# B&R Automation Studio project DevOpsDemo
Automation Studio 6.7.1.5; technology packages: mappMotion 6.7.2, mappView 6.7.0, OpcUaCs 6.6.1

## Configuration Config1

CPU X20CP0484, AutomationRuntime 6.7.5, Build 11.3.0

CPU X20CP1686X, AutomationRuntime 6.7.6, Build 11.3.0

### Task classes (Cpu.sw)
```
Cyclic#1 (cycle 1000 us, tolerance 0 us):
  Program <- Program.prg
  RevInfo <- RevInfo.RevInfo.prg
```

### Task classes (Cpu.sw)
```
Cyclic#1 (cycle 1000 us, tolerance 0 us):
  Main <- Main.Main.prg
  EM_Conveyo <- EM_Conveyor.EM_Conveyor.prg
  EM_Filler <- EM_Filler.EM_Filler.prg
  EM_Capper <- EM_Capper.EM_Capper.prg
Cyclic#3 (cycle 50000 us, tolerance 50000000 us):
  Update <- Services.Update.prg
  RevInfo <- RevInfo.RevInfo.prg
Binaries: udbdef, FWRules, TCData, sysconf, iomap, ashwd, BRRole, asfw, arconfig, ashwac, UaCsConfig
Libraries: MpBase, UaCore, AsIecCon, ArProject, runtime, FileIO, sys_lib, brsystem, BrdkPackML, PackMLCore, MpAlarmX, astime, McBase, McAxis, MpAxis, McAcpAx, McAcpPar, standard, AsIODiag, MpServer
```

### Hardware
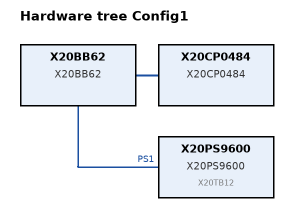
```
X20BB62 : X20BB62 v1.3.0.0
X20CP0484 : X20CP0484 v1.9.0.0  [SL -> X20BB62.SL1]
  Connector IF2:
    ActivateDevice = 1
    Mode = Manual
    InternetAddress = 192.168.2.11
    SubnetMask = 255.255.255.0
    ActivateSnmp = 2
  ConfigurationID = DevOpsDemo_Config1
  UserPartitionSize = 100
  Simulation = 1
  TimerDeviceType = SWIOTIMER
  CyclicTaskClassCount = 3
  Cyclic1Duration = 1000
  Cyclic1Tolerance = 0
  Cyclic2Duration = 5000
  Cyclic2Tolerance = 0
  Cyclic3Duration = 50000
  Cyclic3Tolerance = 50000000
  Cyclic4Duration = 100000
  Cyclic4Tolerance = 100000
  Cyclic5Duration = 200000
  Cyclic5Tolerance = 200000
  Cyclic6Duration = 500000
  Cyclic6Tolerance = 500000
  Cyclic7Duration = 1000000
  Cyclic7Tolerance = 1000000
  Cyclic8Duration = 10000
  Cyclic8Tolerance = 30000000
  FileDevice1
  FileDeviceName1 = USER
  FileDevicePath1 = USER_PATH
  ActivateWebServer = 1
  WebServerProtocol = 1
  ActivateSdm = 1
  Authentication = 0
  ConfigVersion = 0.0.4
X20PS9600 : X20PS9600 v1.6.2.0  [PS -> X20BB62.PS1; SS1 -> X20TB12.SS]
X20TB12 : X20TB12 v1.0.0.0
```

### Config_1.axis - X20CP0484/mappMotion/Config_1.axis
```
Element gAxis_Infeed (Type=axis)
  BaseType = Linear
Element gAxis_Capper (Type=axis)
  BaseType = Rotary
Element gAxis_Outfeed (Type=axis)
  BaseType = Linear
```

### Config.mpbackupcore - X20CP0484/mappServices/Config.mpbackupcore
```
Element gBackupCore (Type=mpbackupcore)
  mapp.Gen:
    Enable = TRUE
    EnableCockpit = FALSE
    Audit = FALSE
    Parent
  Backup:
    AutomaticBackup = Disabled
    AutomaticUpdate = Notify
      DeviceName = UPDATE
      Check = OnEnable
  Alarms = None
```

### Config_1.axis - X20CP1686X/mappMotion/Config_1.axis
```
Element gAxis_Conveyor (Type=axis)
  BaseType = Linear
Element gAxis_Capper (Type=axis)
  MovementLimits:
    Velocity:
      Velocity = 3000
```

## Logical view

Binary libraries used (declarations not repeated): operator, runtime, AsIecCon, MpBase, ArProject, FileIO, sys_lib, brsystem, MpAlarmX, astime, McBase, McAxis, MpAxis, McAcpAx, McAcpPar, standard, AsIODiag, MpServer, AsHttp

### Global.var - Global variables
```iecst
VAR
	gVar : USINT;
END_VAR
```

### Package Logical/Libraries - Global libraries

### Library Logical/Libraries/BrdkPackML (ANSIC, version 3.0.3) - OMAC PackML
Depends on: sys_lib, brsystem

#### BrdkPackML.fun
```iecst
FUNCTION_BLOCK ControlModule (*Control module implementation for OMAC PackML*)
	VAR_INPUT
		Setup : CMSetupType; (*Local setup*) (* *) (*#PAR#;*)
		Interface : CMInterfaceType; (*Publish/Subscribe Interface between Equipment Modules *)
		StateInfo : STRING[255]; (*Status of what the substate is doing or waiting for. Will also be used for logging.*) (* *) (*#CYC#;*)
		State : DINT; (*Control Module state*)
		SubState : DINT := 0; (*The sub state of the module. Can be used for programming the sequence inside a PackML state. Will automatically be reset to 0 by a PackML state change.*) (* *) (*#CYC#;*)
		Continue : BOOL; (*Continue / Acknowledge a state or substate change request when StepMode is enabled*)
	END_VAR
	VAR_OUTPUT
		Info : CMInfoType; (*Additional information about the component*) (* *) (*#CMD#; *)
	END_VAR
	VAR
		Internal : CMInternalType; (*Internal variables*)
	END_VAR
END_FUNCTION_BLOCK

FUNCTION_BLOCK EquipmentModule (*Synchronized PackML state machine handling*) (* $GROUP=mapp Services,$CAT=OMAC PackML,$GROUPICON=Icon_mapp.png,$CATICON=Icon_MpPackML.png *)
	VAR_INPUT
		Setup : EMSetupType; (*Local setup*) (* *) (*#PAR#;*)
		Interface : EMInterfaceType; (*Publish/Subscribe Interface between Equipment Modules *)
		SetModeID : DINT := 1; (*Change the packML mode*)
		StateInfo : STRING[255]; (*Status of what the substate is doing or waiting for. Will also be used for logging.*) (* *) (*#CYC#;*)
		Command : EMCommandType; (*Control commands from ISA-TR88.00.02 commands.*) (* *) (*#CMD#;*)
		SubState : DINT := 0; (*The sub state of the module. Can be used for programming the sequence inside a PackML state. Will automatically be reset to 0 by a PackML state change.*) (* *) (*#CYC#;*)
		Continue : BOOL; (*Continue / Acknowledge a substate change request when StepMode is enabled*)
	END_VAR
	VAR_OUTPUT
		StateCurrent : EMPackMLStateEnum := STATE_UNDEFINED; (*Current state*) (* *) (*#CMD#;*)
		ModeID : EMPackMLModeEnum := MODE_PRODUCTION; (*The current mode*) (* *) (*#CMD#;*)
		Info : EMInfoType; (*Additional information about the component*) (* *) (*#CMD#; *)
	END_VAR
	VAR
		Internal : EMInternalType; (*Internal variables*)
	END_VAR
END_FUNCTION_BLOCK

FUNCTION EMGetModuleAdrByIdx : UDINT (*Returns the address of an Equipment Module on the heap based on the index*)
	VAR_INPUT
		EmIdx : UDINT; (*Index of the Equipment Module*)
	END_VAR
END_FUNCTION

FUNCTION EMGetModuleIdxByName : UDINT (*Returns the index for an Em with the specified name*)
	VAR_INPUT
		EmName : STRING[255]; (*Name of the Equipment Module*)
	END_VAR
END_FUNCTION

FUNCTION EMGetModuleAdrByName : UDINT (*Returns the address of an Equipment Module on the heap based on its name*)
	VAR_INPUT
		EmName : STRING[255]; (*Name of the Equipment Module*)
	END_VAR
END_FUNCTION

FUNCTION EMGetNumberOfModules : UDINT (*Returns the number of Equipment Modules*)
END_FUNCTION

FUNCTION EMGetNumberOfRootModules : UDINT (*Returns the number of root modules. A root module is an Equipment Module with Level 0*)
END_FUNCTION

FUNCTION EMGetWaitingForByIdx : BOOL (*Get WaitingFor from hierarchy index. Returns true on success*)
	VAR_INPUT
		EmIdx : UDINT; (*Index of the root*)
		WaitingFor : EMStatusType; (*EMStatusType*)
	END_VAR
END_FUNCTION

FUNCTION EMGetInterruptedByByIdx : BOOL (*Get InterruptedBy from hierarchy index. Returns true on success*)
	VAR_INPUT
		EmIdx : UDINT; (*Index of the root*)
		InterruptedBy : EMStatusType; (*EMStatusType*)
	END_VAR
END_FUNCTION

FUNCTION EMGetModuleStatus : BOOL (*Get the status from any Equipment Module using the memory address. Returns true on success*)
	VAR_INPUT
		EmAddress : UDINT; (*Address of the Equipment Module*)
		EMStatus : EMStatusType; (*EMStatusType*)
	END_VAR
END_FUNCTION

FUNCTION EMGetModuleStatusByName : BOOL (*Get the status from any Equipment Module using the configured name. Returns true on success*)
	VAR_INPUT
		EmName : STRING[255]; (*Name of the Equipment Module*)
		EMStatus : EMStatusType; (*EMStatusType*)
	END_VAR
END_FUNCTION

FUNCTION EMGetModuleStatusByIdx : BOOL (*Get the status from any Equipment Module using an index. Returns true on success*)
	VAR_INPUT
		EmIdx : UDINT; (*Index of the Equipment Module*)
		EMStatus : EMStatusType; (*EMStatusType*)
	END_VAR
END_FUNCTION

FUNCTION EMGetParentAdr : UDINT (*Returns the address of the parent Equipment Module on the heap*)
	VAR_INPUT
		EmAddress : UDINT; (*Address of the Equipment Module*)
	END_VAR
END_FUNCTION

FUNCTION EMGetChildrenAdrByIdx : UDINT (*Returns the address of a child Equipment Module using an index*)
	VAR_INPUT
		EmAddress : UDINT; (*Address of the Equipment Module*)
		EmIdx : UDINT; (*Index of the child Equipment Module*)
	END_VAR
END_FUNCTION

FUNCTION EMGetSiblingAdrByIdx : UDINT (*Returns the address of a sibling Equipment Module using an index*)
	VAR_INPUT
		EmAddress : UDINT; (*Address of the Equipment Module*)
		EmIdx : UDINT; (*Index of the sibling Equipment Module*)
	END_VAR
END_FUNCTION

FUNCTION EMGetRootAdrByIdx : UDINT (*Returns the address of a root Equipment Module using an index*)
	VAR_INPUT
		EmIdx : UDINT; (*Index of a root Equipment Module*)
	END_VAR
END_FUNCTION

FUNCTION EMGetUserDataAdr : UDINT (*Returns the address of the published userdata from a remote Equipment Module*)
	VAR_INPUT
		EmAddress : UDINT; (*Address of the Equipment Module*)
	END_VAR
END_FUNCTION

FUNCTION EMSetCommand : BOOL (*Send a command to an Equipment Module using its address. Returns true on success*)
	VAR_INPUT
		EmAddress : UDINT; (*Address of the remote Equipment Module to receive the command*)
		EmAddressInterrupter : UDINT; (*Address of the local Equipment Module interrupting the remote Em *)
		Command : EMPackMLCmdEnum; (*Command*)
	END_VAR
END_FUNCTION

FUNCTION EMSetMode : BOOL (*Function changing the mode of an Equipment Module*) (* $GROUP=mapp Services,$CAT=OMAC PackML,$GROUPICON=Icon_mapp.png,$CATICON=Icon_MpPackML.png *)
	VAR_INPUT
		EmAddress : UDINT; (*Address of the target Equipment Module*)
		Mode : DINT; (*Desired mode to change to. The mode must be defined in the mppackmlcore configuration*) (* *) (*#PAR#;*)
	END_VAR
END_FUNCTION

FUNCTION EMSetModeByName : BOOL (*Function changing the mode of an Equipment Module*) (* $GROUP=mapp Services,$CAT=OMAC PackML,$GROUPICON=Icon_mapp.png,$CATICON=Icon_MpPackML.png *)
	VAR_INPUT
		EmName : STRING[255]; (*Name of the target Equipment Module*)
		Mode : DINT; (*Desired mode to change to. *) (* *) (*#PAR#;*)
	END_VAR
END_FUNCTION
```

#### BrdkPackML.typ
```iecst
TYPE
	EMStatusType : 	STRUCT  (*EMStatusType*)
		Name : STRING[255]; (*Em Name*)
		ModeID : UDINT; (*Current Mode*)
		StateCurrent : EMPackMLStateEnum; (*Current State*)
		SubStateCurrent : DINT; (*Current Sub State*)
		StateComplete : BOOL; (*State Complete*)
		StateInfo : STRING[255]; (*Used to describe the action in all states and substates*)
	END_STRUCT;
	EMCommandType : 	STRUCT  (*EMCommandType*)
		Abort : BOOL; (*Go to state Aborting - Can be set in all states except Aborting and Aborted.*)
		Clear : BOOL; (*Go to state Clearing - Can only be set in state Aborted.*)
		Stop : BOOL; (*Go to state Stopping - Can be set in all states except Aborting, Aborted, Clearing, Stopping and Stopped.*)
		Reset : BOOL; (*Go to state Resetting - Can only be set in state Stopped.*)
		Start : BOOL; (*Go to state Starting - Can only be set in state Idle.*)
		Hold : BOOL; (*Go to state Holding. Can only be set in state Execute.*)
		Unhold : BOOL; (*Go to state Unholding. Can only be set in state Held.*)
		Suspend : BOOL; (*Go to state Suspending. Can only be set in state Execute.*)
		Unsuspend : BOOL; (*Go to state Unsuspending. Can only be set in state Suspended.*)
		Complete : BOOL; (*Go to state Completing. Can only be set in state Execute*)
		StateComplete : BOOL; (*Go to next waiting state. Can be set in all acting states and state Execute.*)
	END_STRUCT;
	EMPackMLCmdEnum :
		( (*Command Enum*)
		CMD_UNDEFINED := 0, (*Undefined Command*)
		CMD_RESET := 1, (*PackML Reset Command*)
		CMD_START := 2, (*PackML Start Command*)
		CMD_STOP := 3, (*PackML Stop Command*)
		CMD_HOLD := 4, (*PackML Hold Command*)
		CMD_UNHOLD := 5, (*PackML Unhold Command*)
		CMD_SUSPEND := 6, (*PackML Suspend Command*)
		CMD_UNSUSPEND := 7, (*PackML Unsuspend Command*)
		CMD_ABORT := 8, (*PackML Abort Command*)
		CMD_CLEAR := 9, (*PackML Clear Command*)
		CMD_COMPLETE := 10, (*PackML Complete Command*)
		CMD_SC := 11 (*PackML State Complete Command*)
		);
	EMPackMLModeEnum :
		( (*Mode Enum*)
		MODE_UNDEFINED := 0, (*PackML Undefined mode*)
		MODE_PRODUCTION := 1, (*PackML Production mode*)
		MODE_MAINTENANCE := 2, (*PackML Maintenance mode*)
		MODE_MANUAL := 3, (*PackML Manual mode*)
		MODE_CLEAN := 16, (*PackML Cleaning mode*)
		MODE_JOG := 17, (*PackML Jogging mode*)
		MODE_CIP := 18, (*PackML CIP mode*)
		MODE_CALIBRATION := 19 (*PackML Calibration mode*)
		);
	EMPackMLStateEnum :
		( (*State Enum*)
		STATE_UNDEFINED := 0, (*The system is inactive, no state active*)
		STATE_CLEARING := 1, (*PackML CLEARING state*)
		STATE_STOPPED := 2, (*PackML STOPPED state*)
		STATE_STARTING := 3, (*PackML STARTING state*)
		STATE_IDLE := 4, (*PackML IDLE state*)
		STATE_SUSPENDED := 5, (*PackML SUSPENDED state*)
		STATE_EXECUTE := 6, (*PackML EXECUTE state*)
		STATE_STOPPING := 7, (*PackML STOPPING state*)
		STATE_ABORTING := 8, (*PackML ABORTING state*)
		STATE_ABORTED := 9, (*PackML ABORTED state*)
		STATE_HOLDING := 10, (*PackML HOLDING state*)
		STATE_HELD := 11, (*PackML HELD state*)
		STATE_UNHOLDING := 12, (*PackML UNHOLDING state*)
		STATE_SUSPENDING := 13, (*PackML SUSPENDING state*)
		STATE_UNSUSPENDING := 14, (*PackML UNSUSPENDING state*)
		STATE_RESETTING := 15, (*PackML RESETTING state*)
		STATE_COMPLETING := 16, (*PackML COMPLETING state*)
		STATE_COMPLETED := 17, (*PackML COMPLETED state*)
		STATE_DEACTIVATING := 30, (*Deactivating state. Not a standard PackML state*)
		STATE_DEACTIVATED := 31, (*Deactivated state. Not a standard PackML state*)
		STATE_ACTIVATING := 32 (*Activating state. Not a standard PackML state*)
		);
	EMActivationConditionEnum :
		( (*Activation Enum*)
		ACTIVATE_AUTOMATIC := 0, (*Activate Em automatically when executed*)
		ACTIVATE_BY_PARENT := 1, (*Activate Em if parent is activated*)
		ACTIVATE_BY_PV := 2 (*Activate Em based on PV value*)
		);
	EMSetupType : 	STRUCT  (*EMSetupType*)
		ParentName : STRING[255]; (*Name of the parent. Leave empty is Em is parent at level 0*)
		Name : STRING[255]; (*Name of the Em. If left empty during first execution, the task name is used as Em name*)
		NameIndex : USINT := EM_MAX_NAME_INDEX; (*Index of the Em if having multiple Em's in an array*)
		Activate : BOOL := FALSE; (*PV for ActivationCondition ACTIVATE_BY_PV*)
		ActivationCondition : EMActivationConditionEnum := ACTIVATE_AUTOMATIC; (*Condition for activating the Em*)
		EnableWaitingFor : BOOL := TRUE; (*Enable the WaitingFor log*)
		EnableInterruptedBy : BOOL := TRUE; (*Enable the InterruptedBy log*)
		Synchronization : EMSynchronizationType; (*Parameters for Em synchronization*)
		AuditModeChange : BOOL := TRUE; (*Log when mode is changed*)
		AuditStateChange : BOOL := TRUE; (*Log when state is changed*)
		AuditSubStateChange : BOOL := TRUE; (*Log when substate is changed*)
		SkipStopStateComplete : BOOL; (*The StateComplete command is ignored during stop*)
		StepMode : BOOL; (*Enables StepMode for substate changes*)
	END_STRUCT;
	EMInfoType : 	STRUCT  (*EMInfoType*)
		ParentName : STRING[255]; (*Name of the Parent Em*)
		ParentStateCurrent : EMPackMLStateEnum; (*Parent Current State*)
		EmName : STRING[255]; (*Name of the Em*)
		EmAddress : UDINT; (*Address of the Em*)
		EmIndex : UDINT; (*Global EM index*)
		UserDataAddress : UDINT; (*Published data address*)
		Level : UDINT; (*Level in the hierarchy. Parent is level 0.*)
		SiblingCount : UDINT; (*Number of Siblings. No siblings means Sibling count 1*)
		ChildCount : UDINT; (*How many children are registered to this module. Even when desynchronized the child count will still be valid.*)
		ParentStateComplete : BOOL; (*The parent is state complete. Can be used to synchronize a state transition*)
		SiblingsStateComplete : BOOL; (*All siblings are state complete. Can be used to synchronize a state transition*)
		ChildrenStateComplete : BOOL; (*All children are state complete. Can be used to synchronize a state transition*)
		WaitingFor : EMStatusType; (*The status for the Em we are waiting for*)
		InterruptedBy : EMStatusType; (*The Em we where interrupted by*)
		TimeInState : REAL; (*The actual time in the current state*)
		TimeInSubState : REAL; (*The actual time in the current sub state*)
		Last : ARRAY[0..EM_MAX_AUDIT_ENTRIES]OF STRING[50]; (*The last state, substate and mode*)
		CycleTime : REAL; (*Cycle Time in seconds*)
		OnStateEntry : BOOL; (*Goes to true on the first scan after a state change*)
		OnSubStateEntry : BOOL; (*Goes to true on the first scan after a substate change*)
	END_STRUCT;
	EMInternalType : 	STRUCT  (*Internal type of the Em*)
		state : USINT; (*Internal state*)
		emAddress : UDINT; (*Address of the instance on the heap memory*)
		nextSubState : DINT; (*Next substate when StepMode is enabled*)
		userDataAddress : UDINT; (*Address of the user data on the heap memory*)
		subscriptionUserDataAddress : ARRAY[0..EM_MAX_SUBSCRIPTIONS]OF UDINT; (*Address of the user data we are currently subscribing to*)
		subscribedToEMName : ARRAY[0..EM_MAX_SUBSCRIPTIONS]OF STRING[255]; (*Name of the Em we are subscribed to*)
		oldPubSubEnable : BOOL; (*Old Pub/Sub enable*)
	END_STRUCT;
	EMSynchronizationType : 	STRUCT  (*Em synchronization settings type*)
		Override : EMSynchronizationCmdType := (Abort:=FALSE,Stop:=FALSE,Complete:=FALSE,Suspend:=FALSE,Unsuspend:=FALSE,Hold:=FALSE,Unhold:=TRUE,Clear:=TRUE,Reset:=TRUE,Start:=TRUE); (*Commands that are overriden by parrent command*)
		ReactTo : EMSynchronizationCmdType := (Abort:=TRUE,Stop:=TRUE,Complete:=TRUE,Suspend:=TRUE,Unsuspend:=TRUE,Hold:=TRUE,Unhold:=TRUE,Clear:=TRUE,Reset:=TRUE,Start:=TRUE); (*Commands that are reacted to by parent*)
		Escalate : EMSynchronizationCmdType := (Abort:=TRUE,Stop:=TRUE,Complete:=TRUE,Suspend:=TRUE,Unsuspend:=TRUE,Hold:=TRUE,Unhold:=FALSE,Clear:=FALSE,Reset:=FALSE,Start:=FALSE); (*Commands that are escalated to the parrent*)
	END_STRUCT;
	EMSynchronizationCmdType : 	STRUCT  (*Em synchronization settings type*)
		Abort : BOOL := FALSE; (*Synchronization setting for command*)
		Stop : BOOL := FALSE; (*Synchronization setting for command*)
		Complete : BOOL := FALSE; (*Synchronization setting for command*)
		Suspend : BOOL := FALSE; (*Synchronization setting for command*)
		Unsuspend : BOOL := FALSE; (*Synchronization setting for command*)
		Hold : BOOL := FALSE; (*Synchronization setting for command*)
		Unhold : BOOL := FALSE; (*Synchronization setting for command*)
		Clear : BOOL := FALSE; (*Synchronization setting for command*)
		Reset : BOOL := FALSE; (*Synchronization setting for command*)
		Start : BOOL := FALSE; (*Synchronization setting for command*)
	END_STRUCT;
	EMInterfaceType : 	STRUCT  (*Interface type*)
		Enable : BOOL; (*Enable Pub/Sub interface*)
		SubscriptionEMName : ARRAY[0..EM_MAX_SUBSCRIPTIONS]OF STRING[255]; (*Name of the Em where we want cyclic user data from*)
		SubscriptionValid : ARRAY[0..EM_MAX_SUBSCRIPTIONS]OF BOOL; (*True if data is valid. Only true if Em name does exist*)
		Publish : EMUserDataPubSubType; (*The local user data that other Em can subscribe to*)
		Subscribe : ARRAY[0..EM_MAX_SUBSCRIPTIONS]OF EMUserDataPubSubType; (*The user data from the remote Em that we are subscribing to*)
	END_STRUCT;
END_TYPE

(*CM*)

TYPE
	CMInternalType : 	STRUCT  (*Internal type of the Cm*)
		state : USINT; (*Internal state*)
		parentEmAddress : UDINT; (*Address of the instance on the heap memory*)
		subscriptionUserDataAddress : ARRAY[0..EM_MAX_SUBSCRIPTIONS]OF UDINT; (*Address of the user data we are currently subscribing to*)
		subscribedToEMName : ARRAY[0..EM_MAX_SUBSCRIPTIONS]OF STRING[255]; (*Name of the Em we are subscribed to*)
		oldParentState : DINT; (*Old parent state*)
		oldState : DINT; (*Old state*)
		nextState : DINT; (*Next state when StepMode is enabled*)
		oldSubState : DINT; (*Old sub state*)
		nextSubState : DINT; (*Next substate when StepMode is enabled*)
		cycleTime : REAL; (*Cycle time for the module task class*)
		oldPubSubEnable : BOOL; (*Old Pub/Sub enable*)
	END_STRUCT;
	CMSetupType : 	STRUCT  (*CMSetupType*)
		ParentName : STRING[255]; (*Name of the parent. Leave empty is Em is parent at level 0*)
		Name : STRING[255]; (*Name of the Em. If left empty during first execution, the task name is used as Em name*)
		NameIndex : USINT := EM_MAX_NAME_INDEX;
		AuditStateChange : BOOL := TRUE; (*Log when state is changed*)
		AuditSubStateChange : BOOL := TRUE; (*Log when substate is changed*)
		StepMode : BOOL; (*Enables StepMode for state and substate changes*)
	END_STRUCT;
	CMInfoType : 	STRUCT  (*CMInfoType*)
		CmName : STRING[255]; (*Name of the Cm*)
		ParentName : STRING[255]; (*Name of the Parent Em*)
		ParentEmAddress : UDINT; (*Address of the Em*)
		ParentEmIndex : UDINT; (*Global EM index*)
		ParentStateCurrent : EMPackMLStateEnum; (*Parent Current State*)
		Level : UDINT; (*Level in the hierarchy. Parent is level 0.*)
		TimeInState : REAL; (*The actual time in the current state*)
		TimeInSubState : REAL; (*The actual time in the current sub state*)
		Last : ARRAY[0..EM_MAX_AUDIT_ENTRIES]OF STRING[50]; (*The last state, substate and mode*)
		CycleTime : REAL; (*Cycle Time in seconds*)
		OnStateEntry : BOOL; (*True in first scan after a state change*)
		OnSubStateEntry : BOOL; (*True in first scan after a substate change*)
	END_STRUCT;
	CMInterfaceType : 	STRUCT  (*Interface type*)
		Enable : BOOL; (*Enable Sub interface*)
		SubscriptionEMName : ARRAY[0..EM_MAX_SUBSCRIPTIONS]OF STRING[255]; (*Name of the Em where we want cyclic user data from*)
		SubscriptionValid : ARRAY[0..EM_MAX_SUBSCRIPTIONS]OF BOOL; (*True if data is valid. Only true if Em name does exist*)
		Subscribe : ARRAY[0..EM_MAX_SUBSCRIPTIONS]OF EMUserDataPubSubType; (*The user data from the remote Em that we are subscribing to*)
	END_STRUCT;
END_TYPE

(******* USER DEFINED *******)

TYPE
	EMUserDataPubSubType : 	STRUCT  (*Local / Remote user data. This datatype can be expanded to fit the needs of the application*)
		State : EMPackMLStateEnum;
		SubState : DINT;
		StateComplete : BOOL;
		CmdAbortCounter : UDINT;
		CmdStopCounter : UDINT;
		Priority : UDINT;
		PrioritySC : BOOL;
	END_STRUCT;
END_TYPE
```

#### BrdkPackMLFunctions.cpp
```cpp
#include "BrdkPackML.h"
#include "../PackMLCore/PackMLModule.hpp"
#include "../PackMLCore/PackMLModuleTable.hpp"

unsigned long bur_heap_size = 0x3CCCC;

PackMLModuleTable* pPackMLModuleTable = new PackMLModuleTable();

//---------------------- IEC Functions ----------------------------------//
bool EMSetMode(unsigned long EmAddress, signed long Mode)
{
	if(EmAddress == 0){
		return false;
	}

	PackMLModule* pPackMLModule = reinterpret_cast<PackMLModule*>(EmAddress);

	return pPackMLModule->setCurrentMode(Mode);

}

bool EMSetModeByName(plcstring* EmName, signed long Mode)
{
	PackMLModule* pPackMLModule = pPackMLModuleTable->getModuleByName(EmName);

	if(pPackMLModule == nullptr)
		return false;

	return pPackMLModule->setCurrentMode(Mode);

}

plcbit EMGetModuleStatusByName(plcstring* EmName, struct EMStatusType* EMStatus){

	PackMLModule* pPackMLModule = pPackMLModuleTable->getModuleByName(EmName);

	if(EMStatus == 0 || pPackMLModule == nullptr){
		return false;
	}

	EMStatus->ModeID = pPackMLModule->getCurrentMode();
	strcpy(EMStatus->Name, pPackMLModule->getModuleName());
	EMStatus->StateComplete = pPackMLModule->getStateComplete();
	EMStatus->StateCurrent = static_cast<EMPackMLStateEnum>(pPackMLModule->getCurrentState());
	EMStatus->SubStateCurrent = pPackMLModule->getCurrentSubState();
	strcpy(EMStatus->StateInfo, pPackMLModule->getStateInfo());

	return true;
}

plcbit EMGetWaitingForByIdx(unsigned long EmIdx, struct EMStatusType* WaitingFor){

	PackMLModule* pPackMLModule = pPackMLModuleTable->getRootModuleByIdx(EmIdx);

	if(WaitingFor == 0 || pPackMLModule == nullptr){
		return false;
	}

	unsigned long int waitingForIndex =  pPackMLModule->getWaitingForIndex();

	if(waitingForIndex == 0xFFFFFFFF){
		return false;
	}

	PackMLModule* pWaitingFor = pPackMLModuleTable->getModuleByIdx(waitingForIndex);

	WaitingFor->ModeID = pWaitingFor->getCurrentMode();
	WaitingFor->StateCurrent = static_cast<EMPackMLStateEnum>(pWaitingFor->getCurrentState());
	WaitingFor->SubStateCurrent = pWaitingFor->getCurrentSubState();
	WaitingFor->StateComplete = pWaitingFor->getStateComplete();
	strcpy(WaitingFor->Name, pWaitingFor->getModuleName());
	strcpy(WaitingFor->StateInfo, pWaitingFor->getStateInfo());

	return true;
}

plcbit EMGetInterruptedByByIdx(unsigned long EmIdx, struct EMStatusType* InterruptedBy){

	PackMLModule* pPackMLModule = pPackMLModuleTable->getModuleByIdx(EmIdx);

	if(InterruptedBy == 0 || pPackMLModule == nullptr){
		return false;
	}

	unsigned long int interruptedByIndex =  pPackMLModule->getInterruptedByIndex();

	if(interruptedByIndex == 0xFFFFFFFF){
		return false;
	}

	PackMLModule* pInterruptedBy = pPackMLModuleTable->getModuleByIdx(interruptedByIndex);

	InterruptedBy->ModeID = pInterruptedBy->getCurrentMode();
	InterruptedBy->StateCurrent = static_cast<EMPackMLStateEnum>(pInterruptedBy->getInterruptedInState());
	InterruptedBy->SubStateCurrent = pInterruptedBy->getInterruptedInSubState();
	InterruptedBy->StateComplete = false;
	strcpy(InterruptedBy->Name, pInterruptedBy->getModuleName());

	//			strcpy(inst->Info.InterruptedBy.StateInfo, pInterruptedBy->getStateInfo());
	return true;
}

unsigned long EMGetModuleAdrByName(plcstring* EmName){

	return reinterpret_cast<unsigned long int>(pPackMLModuleTable->getModuleByName(EmName));
}

unsigned long EMGetModuleAdrByIdx(unsigned long EmIdx){

	return reinterpret_cast<unsigned long int>(pPackMLModuleTable->getModuleByIdx(EmIdx));
}

plcbit EMGetModuleStatus(unsigned long EmAddress, struct EMStatusType* EMStatus){

	if(EmAddress == 0 || EMStatus == 0){
		return false;
	}

	PackMLModule* pPackMLModule = reinterpret_cast<PackMLModule*>(EmAddress);

	EMStatus->ModeID = pPackMLModule->getCurrentMode();
	strcpy(EMStatus->Name, pPackMLModule->getModuleName());
	EMStatus->StateComplete = pPackMLModule->getStateComplete();
	EMStatus->StateCurrent = static_cast<EMPackMLStateEnum>(pPackMLModule->getCurrentState());
	EMStatus->SubStateCurrent = pPackMLModule->getCurrentSubState();
	strcpy(EMStatus->StateInfo, pPackMLModule->getStateInfo());

	return true;
}

unsigned long EMGetNumberOfModules(){
	return pPackMLModuleTable->getNumberOfModules();
}

unsigned long EMGetNumberOfRootModules(){
	return pPackMLModuleTable->getNumberOfRoots();
}

plcbit EMGetModuleStatusByIdx(unsigned long EmIdx, struct EMStatusType* EMStatus){

	if(EMStatus == 0){
		return false;
	}

	PackMLModule* pPackMLModule = pPackMLModuleTable->getModuleByIdx(EmIdx);

	EMStatus->ModeID = pPackMLModule->getCurrentMode();
	strcpy(EMStatus->Name, pPackMLModule->getModuleName());
	EMStatus->StateComplete = pPackMLModule->getStateComplete();
	EMStatus->StateCurrent = static_cast<EMPackMLStateEnum>(pPackMLModule->getCurrentState());
	EMStatus->SubStateCurrent = pPackMLModule->getCurrentSubState();
	strcpy(EMStatus->StateInfo, pPackMLModule->getStateInfo());

	return true;
}

unsigned long EMGetParentAdr(unsigned long EmAddress){

	if(EmAddress == 0){
		return 0;
	}
	return reinterpret_cast<unsigned long int>(reinterpret_cast<PackMLModule*>(EmAddress)->getParentPtr());
		}
unsigned long EMGetChildrenAdrByIdx(unsigned long EmAddress, unsigned long EmIdx){

	if(EmAddress == 0){
		return 0;
	}

	return reinterpret_cast<unsigned long int>(reinterpret_cast<PackMLModule*>(EmAddress)->getChildPtr(EmIdx));

		}
unsigned long EMGetSiblingAdrByIdx(unsigned long EmAddress, unsigned long EmIdx){

	if(EmAddress == 0){
		return 0;
	}

	return reinterpret_cast<unsigned long int>(reinterpret_cast<PackMLModule*>(EmAddress)->getSiblingPtr(EmIdx));

		}
unsigned long EMGetRootAdrByIdx(unsigned long EmIdx){

	return reinterpret_cast<unsigned long int>(pPackMLModuleTable->getRootModuleByIdx(EmIdx));

}
unsigned long EMGetUserDataAdr(unsigned long EmAddress){

	if(EmAddress == 0){
		return 0;
	}
	return reinterpret_cast<unsigned long int>(reinterpret_cast<PackMLModule*>(EmAddress)->getUserMemoryPtr());

		}

plcbit EMSetCommand(unsigned long EmAddress, unsigned long EmAddressInterrupter, enum EMPackMLCmdEnum Command){

	if(EmAddress == 0){
		return false;
	}

	PackMLModule* pPackMLModule = reinterpret_cast<PackMLModule*>(EmAddress);
	PackMLModuleStateEnu cmdState;

	switch(Command){

		case CMD_ABORT:
			pPackMLModule->setCmdAbort();
			cmdState = ST_ABORTING;
			break;

		case CMD_STOP:
			pPackMLModule->setCmdStop();
			cmdState = ST_STOPPING;
			break;

		case CMD_CLEAR:
			pPackMLModule->setCmdClear();
			cmdState = ST_CLEARING;
			break;

		case CMD_RESET:
			pPackMLModule->setCmdReset();
			cmdState = ST_RESETTING;
			break;

		case CMD_START:
			pPackMLModule->setCmdStart();
			cmdState = ST_STARTING;
			break;

		case CMD_HOLD:
			pPackMLModule->setCmdHold();
			cmdState = ST_HOLDING;
			break;

		case CMD_UNHOLD:
			pPackMLModule->setCmdUnhold();
			cmdState = ST_UNHOLDING;
			break;

		case CMD_SUSPEND:
			pPackMLModule->setCmdSuspend();
			cmdState = ST_SUSPENDING;
			break;

		case CMD_UNSUSPEND:
			pPackMLModule->setCmdUnsuspend();
			cmdState = ST_UNSUSPENDING;
			break;

		case CMD_COMPLETE:
			pPackMLModule->setCmdComplete();
			cmdState = ST_COMPLETING;
			break;

		case CMD_SC:
			pPackMLModule->setCmdStateComplete();
			cmdState = ST_UNDEFINED;
			break;

		default:
			return false;

	}

	if(EmAddressInterrupter != 0 && Command != CMD_SC){
		pPackMLModule->setInterruptedBy(reinterpret_cast<PackMLModule*>(EmAddressInterrupter), cmdState);
	}

	return true;

}

unsigned long EMGetModuleIdxByName(plcstring* EmName){

	if(EmName == nullptr){
		return 0xFFFFFFFF;
	}

	return pPackMLModuleTable->getModuleIndexByName(EmName);

}
```

#### EquipmentModule.cpp
```cpp
#include "BrdkPackML.h"
#include "../PackMLCore/PackMLModule.hpp"
#include "../PackMLCore/PackMLModuleTable.hpp"

extern unsigned long bur_heap_size;

extern PackMLModuleTable* pPackMLModuleTable;

// Main function. Is running cyclic together with FUB EquipmentModule()
void run(struct EquipmentModule* inst, PackMLModule* pPackMLModule)
{
	// Reading Setup structure
	pPackMLModule->setActivationCondition(static_cast<short int>(inst->Setup.ActivationCondition));
	pPackMLModule->setActivationPv(inst->Setup.Activate);

	pPackMLModule->setOverrideAbort(inst->Setup.Synchronization.Override.Abort);
	pPackMLModule->setOverrideStop(inst->Setup.Synchronization.Override.Stop);
	pPackMLModule->setOverrideComplete(inst->Setup.Synchronization.Override.Complete);
	pPackMLModule->setOverrideSuspend(inst->Setup.Synchronization.Override.Suspend);
	pPackMLModule->setOverrideUnsuspend(inst->Setup.Synchronization.Override.Unsuspend);
	pPackMLModule->setOverrideHold(inst->Setup.Synchronization.Override.Hold);
	pPackMLModule->setOverrideUnhold(inst->Setup.Synchronization.Override.Unhold);
	pPackMLModule->setOverrideClear(inst->Setup.Synchronization.Override.Clear);
	pPackMLModule->setOverrideReset(inst->Setup.Synchronization.Override.Reset);
	pPackMLModule->setOverrideStart(inst->Setup.Synchronization.Override.Start);

	pPackMLModule->setReactToAbort(inst->Setup.Synchronization.ReactTo.Abort);
	pPackMLModule->setReactToStop(inst->Setup.Synchronization.ReactTo.Stop);
	pPackMLModule->setReactToComplete(inst->Setup.Synchronization.ReactTo.Complete);
	pPackMLModule->setReactToSuspend(inst->Setup.Synchronization.ReactTo.Suspend);
	pPackMLModule->setReactToUnsuspend(inst->Setup.Synchronization.ReactTo.Unsuspend);
	pPackMLModule->setReactToHold(inst->Setup.Synchronization.ReactTo.Hold);
	pPackMLModule->setReactToUnhold(inst->Setup.Synchronization.ReactTo.Unhold);
	pPackMLModule->setReactToClear(inst->Setup.Synchronization.ReactTo.Clear);
	pPackMLModule->setReactToReset(inst->Setup.Synchronization.ReactTo.Reset);
	pPackMLModule->setReactToStart(inst->Setup.Synchronization.ReactTo.Start);

	pPackMLModule->setEscalateAbort(inst->Setup.Synchronization.Escalate.Abort);
	pPackMLModule->setEscalateStop(inst->Setup.Synchronization.Escalate.Stop);
	pPackMLModule->setEscalateComplete(inst->Setup.Synchronization.Escalate.Complete);
	pPackMLModule->setEscalateSuspend(inst->Setup.Synchronization.Escalate.Suspend);
	pPackMLModule->setEscalateUnsuspend(inst->Setup.Synchronization.Escalate.Unsuspend);
	pPackMLModule->setEscalateHold(inst->Setup.Synchronization.Escalate.Hold);
	pPackMLModule->setEscalateUnhold(inst->Setup.Synchronization.Escalate.Unhold);
	pPackMLModule->setEscalateClear(inst->Setup.Synchronization.Escalate.Clear);
	pPackMLModule->setEscalateReset(inst->Setup.Synchronization.Escalate.Reset);
	pPackMLModule->setEscalateStart(inst->Setup.Synchronization.Escalate.Start);

	if (inst->Info.OnStateEntry){
		inst->Info.OnStateEntry = false;
	}
	if (inst->Info.OnSubStateEntry){
		inst->Info.OnSubStateEntry = false;
	}

	long int oldSubstate = pPackMLModule->getCurrentSubState();

	if(oldSubstate == -1){
		inst->SubState = -1;

		if(inst->Continue || !inst->Setup.StepMode){
			inst->SubState = inst->Internal.nextSubState;
			pPackMLModule->setCurrentSubState(inst->SubState);
			inst->Info.OnSubStateEntry = true;
			inst->Internal.nextSubState = 0;
			inst->Continue = false;
			inst->StateInfo[0] = 0;
		}

	} else if(oldSubstate != inst->SubState){
		if(inst->Setup.AuditSubStateChange){

			for(unsigned short int i = 0; i < EM_MAX_AUDIT_ENTRIES; i++){
				strcpy(inst->Info.Last[EM_MAX_AUDIT_ENTRIES - i], inst->Info.Last[(EM_MAX_AUDIT_ENTRIES - 1) - i]);
			}
			sprintf(inst->Info.Last[0], "Substate: %ld, time: %2.1f s.", oldSubstate, inst->Info.TimeInSubState);
		}

		if(inst->Setup.StepMode && !inst->Continue){
			inst->Internal.nextSubState = inst->SubState;
			sprintf(inst->StateInfo, "Waiting for continue cmd. Next Substate: %ld", inst->Internal.nextSubState);
			inst->SubState = -1;
			pPackMLModule->setCurrentSubState(inst->SubState);
			inst->Continue = false;
		} else {
			pPackMLModule->setCurrentSubState(inst->SubState);
			inst->StateInfo[0] = 0;
			inst->Info.OnSubStateEntry = true;
			inst->Continue = false;
		}

	}

	std::string oldStateInfo = pPackMLModule->getStateInfo();
	if(oldStateInfo != inst->StateInfo){
		pPackMLModule->setStateInfo(inst->StateInfo);
	}

	if(inst->SetModeID != inst->ModeID){
		// Restrict mode changes to certain states could be defined here: (-And also in the function EMSetMode())
		if (!pPackMLModule->setCurrentMode(inst->SetModeID)){
			inst->SetModeID = inst->ModeID;
		}

	}

	pPackMLModule->evaluateCmdAbort(inst->Command.Abort);
	pPackMLModule->evaluateCmdStop(inst->Command.Stop);
	pPackMLModule->evaluateCmdClear(inst->Command.Clear);
	pPackMLModule->evaluateCmdReset(inst->Command.Reset);
	pPackMLModule->evaluateCmdStart(inst->Command.Start);
	pPackMLModule->evaluateCmdSuspend(inst->Command.Suspend);
	pPackMLModule->evaluateCmdUnsuspend(inst->Command.Unsuspend);
	pPackMLModule->evaluateCmdHold(inst->Command.Hold);
	pPackMLModule->evaluateCmdUnhold(inst->Command.Unhold);
	pPackMLModule->evaluateCmdComplete(inst->Command.Complete);
	pPackMLModule->evaluateCmdStateComplete(inst->Command.StateComplete);

	if(inst->Setup.SkipStopStateComplete && pPackMLModule->getCmdStop()){
		pPackMLModule->setCmdStateComplete();
	}

	//--- End of things to handle before EM is being executed from lib on heap ---//

	// Run the packmlmodule service
	pPackMLModule->runPackMLModule();

	EMPackMLStateEnum stateCurrent = static_cast<EMPackMLStateEnum>(pPackMLModule->getCurrentState());
	// Update the FB info
	// State info
	if (inst->StateCurrent != stateCurrent) {

		if(inst->Setup.AuditStateChange){
			plcstring* oldStateStr = (plcstring*)pPackMLModule->getStateStr(static_cast<PackMLModuleStateEnu>(inst->StateCurrent));

			for(unsigned short int i = 0; i < EM_MAX_AUDIT_ENTRIES; i++){
				strcpy(inst->Info.Last[EM_MAX_AUDIT_ENTRIES - i], inst->Info.Last[(EM_MAX_AUDIT_ENTRIES - 1) - i]);
			}
			sprintf(inst->Info.Last[0], "State: %s, time: %2.1f s.", oldStateStr, inst->Info.TimeInState);
		}

		inst->StateCurrent = stateCurrent;

		inst->SubState = 0;
		pPackMLModule->setCurrentSubState(inst->SubState);
		inst->StateInfo[0] = 0;
		inst->Info.OnStateEntry = true;
		inst->Info.OnSubStateEntry = true;
		inst->Continue = false;
		inst->Setup.StepMode = false;

		// Reset Cmds
		memset(&inst->Command, 0, sizeof(inst->Command));

	}

	inst->Info.TimeInState = pPackMLModule->getTimeInState();
	inst->Info.TimeInSubState = pPackMLModule->getTimeInSubState();

	inst->Info.ParentStateCurrent = static_cast<EMPackMLStateEnum>(pPackMLModule->getParentCurrentState());

	// Parent / Child / Sibling state/substate info
	inst->Info.ParentStateComplete = pPackMLModule->getParentStateComplete();
	inst->Info.SiblingsStateComplete = pPackMLModule->getSiblingsStateComplete();
	inst->Info.ChildrenStateComplete = pPackMLModule->getChildrenStateComplete();

	inst->Info.Level = pPackMLModule->getHierarchyLevel();
	inst->Info.ChildCount = pPackMLModule->getChildCount();
	inst->Info.SiblingCount = pPackMLModule->getSiblingCount();

	// Mode info
	if (inst->ModeID != pPackMLModule->getCurrentMode()) {

		if(inst->Setup.AuditStateChange){

			for(unsigned short int i = 0; i < EM_MAX_AUDIT_ENTRIES; i++){
				strcpy(inst->Info.Last[EM_MAX_AUDIT_ENTRIES - i], inst->Info.Last[(EM_MAX_AUDIT_ENTRIES - 1) - i]);
			}
			sprintf(inst->Info.Last[0], "ModeID: %d --> %ld", inst->ModeID, pPackMLModule->getCurrentMode());
		}

		inst->ModeID = static_cast<EMPackMLModeEnum>(pPackMLModule->getCurrentMode());
		inst->SetModeID = inst->ModeID ;

		inst->SubState = 0;
		inst->Continue = false;
		inst->Setup.StepMode = false;
		pPackMLModule->setCurrentSubState(inst->SubState);
		inst->StateInfo[0] = 0;
	}

	if(inst->Setup.EnableInterruptedBy){
		unsigned long int interruptedByIndex =  pPackMLModule->getInterruptedByIndex();
		if(interruptedByIndex != 0xFFFFFFFF){

			PackMLModule* pInterruptedBy = pPackMLModuleTable->getModuleByIdx(interruptedByIndex);

			inst->Info.InterruptedBy.ModeID = inst->ModeID;
			inst->Info.InterruptedBy.StateCurrent = static_cast<EMPackMLStateEnum>(pInterruptedBy->getInterruptedInState());
			inst->Info.InterruptedBy.SubStateCurrent = pInterruptedBy->getInterruptedInSubState();
			inst->Info.InterruptedBy.StateComplete = false;
			strcpy(inst->Info.InterruptedBy.Name, pInterruptedBy->getModuleName());
//			strcpy(inst->Info.InterruptedBy.StateInfo, pInterruptedBy->getStateInfo());
		} else {
			inst->Info.InterruptedBy.ModeID = 0;
			inst->Info.InterruptedBy.StateCurrent = STATE_UNDEFINED;
			inst->Info.InterruptedBy.SubStateCurrent = 0;
			inst->Info.InterruptedBy.StateComplete = false;
			inst->Info.InterruptedBy.Name[0] = 0;
			inst->Info.InterruptedBy.StateInfo[0] = 0;
		}
	}

	if(inst->Setup.EnableWaitingFor){
		unsigned long int waitingForIndex =  pPackMLModule->getWaitingForIndex();
		if(waitingForIndex != 0xFFFFFFFF){

			PackMLModule* pWaitingFor = pPackMLModuleTable->getModuleByIdx(waitingForIndex);

			inst->Info.WaitingFor.ModeID = inst->ModeID;
			inst->Info.WaitingFor.StateCurrent = static_cast<EMPackMLStateEnum>(pWaitingFor->getCurrentState());
			inst->Info.WaitingFor.SubStateCurrent = pWaitingFor->getCurrentSubState();
			inst->Info.WaitingFor.StateComplete = pWaitingFor->getStateComplete();
			strcpy(inst->Info.WaitingFor.Name, pWaitingFor->getModuleName());
			strcpy(inst->Info.WaitingFor.StateInfo, pWaitingFor->getStateInfo());
		} else {
			inst->Info.WaitingFor.ModeID = 0;
			inst->Info.WaitingFor.StateCurrent = STATE_UNDEFINED;
			inst->Info.WaitingFor.SubStateCurrent = 0;
			inst->Info.WaitingFor.StateComplete = false;
			inst->Info.WaitingFor.Name[0] = 0;
			inst->Info.WaitingFor.StateInfo[0] = 0;
		}
	}

	if(inst->Interface.Enable){
		inst->Internal.oldPubSubEnable = true;

		memcpy(reinterpret_cast<EMUserDataPubSubType*>(inst->Internal.userDataAddress), reinterpret_cast<EMUserDataPubSubType*>(&inst->Interface.Publish), sizeof(EMUserDataPubSubType));

		for(unsigned short int i = 0; i < EM_MAX_SUBSCRIPTIONS + 1; i++){

			if(inst->Interface.SubscriptionValid[i]){
				memcpy(reinterpret_cast<EMUserDataPubSubType*>(&inst->Interface.Subscribe[i]), reinterpret_cast<EMUserDataPubSubType*>(inst->Internal.subscriptionUserDataAddress[i]), sizeof(EMUserDataPubSubType));
			}

			if(strcmp(inst->Interface.SubscriptionEMName[i], inst->Internal.subscribedToEMName[i]) != 0){
				PackMLModule* pSubscribtionEm = pPackMLModuleTable->getModuleByName(inst->Interface.SubscriptionEMName[i]);
				if(pSubscribtionEm != nullptr){
					inst->Internal.subscriptionUserDataAddress[i] = reinterpret_cast<unsigned long int>(pSubscribtionEm->getUserMemoryPtr());
					inst->Interface.SubscriptionValid[i] = true;
					strcpy(inst->Internal.subscribedToEMName[i], inst->Interface.SubscriptionEMName[i]);
				} else {
					inst->Interface.SubscriptionValid[i] = false;
					inst->Internal.subscriptionUserDataAddress[i] = 0;
					inst->Internal.subscribedToEMName[i][0] = 0;
				}

				memset(reinterpret_cast<EMUserDataPubSubType*>(&inst->Interface.Subscribe[i]), 0, sizeof(EMUserDataPubSubType));

			}

		}
	} else if(not inst->Interface.Enable && inst->Internal.oldPubSubEnable){
		inst->Internal.oldPubSubEnable = false;
		memset(reinterpret_cast<EMUserDataPubSubType*>(&inst->Interface.Subscribe), 0, sizeof(EMUserDataPubSubType) * (EM_MAX_SUBSCRIPTIONS + 1));
		memset(reinterpret_cast<bool*>(&inst->Interface.SubscriptionValid), 0, sizeof(bool) * (EM_MAX_SUBSCRIPTIONS + 1));
		memset(reinterpret_cast<unsigned long int*>(&inst->Internal.subscriptionUserDataAddress), 0, sizeof(unsigned long int) * (EM_MAX_SUBSCRIPTIONS + 1));
		memset(reinterpret_cast<char*>(&inst->Internal.subscribedToEMName), 0, 256 * (EM_MAX_SUBSCRIPTIONS + 1));
	}

}

// ------------ IEC Functions and Function Blocks -----------------------------------------

void EquipmentModule(struct EquipmentModule* inst)
{

	// Initialize the module
	switch(inst->Internal.state){

		case 0:
			{
				// get name
				if(strlen(inst->Setup.Name) == 0){
					ST_name(0, inst->Setup.Name, 0);
				}

				char moduleName[256] = {""};

				if (inst->Setup.NameIndex == EM_MAX_NAME_INDEX){
					strcpy(moduleName, inst->Setup.Name);
				} else {
					sprintf(moduleName, "%s%d", inst->Setup.Name, inst->Setup.NameIndex);
				}

				// check if object exists
				PackMLModule* pPackMLModule = pPackMLModuleTable->getModuleByName(moduleName);

				// Create a new module if not exists
				if(pPackMLModule == nullptr){
					RTInfo_typ RTInfo_0;
					RTInfo_0.enable = 1;
					RTInfo(&RTInfo_0);

					pPackMLModule = new PackMLModule(moduleName);
					pPackMLModule->setCycleTime(static_cast<float>(RTInfo_0.cycle_time) * 0.000001);
					inst->Info.CycleTime = static_cast<float>(RTInfo_0.cycle_time) * 0.000001;

					// Create userData for misc usage e.g. sync and priority, and get pointer.
					inst->Internal.userDataAddress = reinterpret_cast<unsigned long int>(pPackMLModule->createUserMemory(sizeof(EMUserDataPubSubType)));
					inst->Internal.state = 20;
				} else {
					// We should copy all the options from the heap to the IEC on stack
					strcpy(inst->Setup.ParentName, pPackMLModule->getParentName());
					strcpy(inst->Info.ParentName, inst->Setup.ParentName);

					inst->Internal.userDataAddress = reinterpret_cast<unsigned long int>(pPackMLModule->getUserMemoryPtr());
					inst->Info.EmIndex = pPackMLModuleTable->getModuleIndexByName(moduleName);
					pPackMLModule->setModuleIndex(inst->Info.EmIndex);

					inst->Internal.state = 40;
				}

				inst->Internal.emAddress = reinterpret_cast<unsigned long int>(pPackMLModule);
				inst->Info.EmAddress = inst->Internal.emAddress;
				inst->Info.UserDataAddress = inst->Internal.userDataAddress;
				strcpy(inst->Info.EmName, moduleName);

			}
			break;

		case 20: // register the object
			if(pPackMLModuleTable->registerEm(inst->Internal.emAddress, &inst->Info.EmIndex)){
				PackMLModule* pPackMLModule = reinterpret_cast<PackMLModule*>(inst->Internal.emAddress);
				pPackMLModule->setModuleIndex(inst->Info.EmIndex);
				inst->Internal.state = 30;
			}
			break;

		case 30: // Init EM phase // interlinking
			{
				PackMLModule* pPackMLModule = reinterpret_cast<PackMLModule*>(inst->Internal.emAddress);

				if(strlen(inst->Setup.ParentName) > 0){
					inst->Internal.state = 35;
				} else {
					pPackMLModule->initModule();
					inst->Internal.state = 40;
				}
				strcpy(inst->Info.ParentName, inst->Setup.ParentName);

				// **** do we need it here?? test
				//				pPackMLModule->runPackMLModule();
			}
			break;

		case 35:
			{
				PackMLModule* pPackMLModule = reinterpret_cast<PackMLModule*>(inst->Internal.emAddress);
				// Can get stucked here --> **inst->Info.ParentName**
				if(strcmp(inst->Setup.ParentName, inst->Info.ParentName) != 0){
					inst->Internal.state = 30;
				} else if(pPackMLModule->initModule(reinterpret_cast<PackMLModule*>(pPackMLModuleTable->getModuleByName(inst->Info.ParentName)))){
					//					strcpy(inst->Info.ParentName, pPackMLModule->getParentName());
					inst->Internal.state = 40;
				}

			}
			break;

		case 40: // run state
			// if EmLinkParent changes reinitilise the module in state 30
			{
				PackMLModule* pPackMLModule = reinterpret_cast<PackMLModule*>(inst->Internal.emAddress);

				if(strcmp(inst->Setup.ParentName, inst->Info.ParentName) != 0){
					inst->Internal.state = 50;
				} else {
					run(inst, pPackMLModule);
				}

			}
			break;

		case 50: // exit module and go to state 10
			{
				PackMLModule* pPackMLModule = reinterpret_cast<PackMLModule*>(inst->Internal.emAddress);

				if(pPackMLModule->exitModule()){
					inst->Internal.state = 30;

					if(inst->Setup.AuditStateChange){
						plcstring* oldStateStr = (plcstring*)pPackMLModule->getStateStr(static_cast<PackMLModuleStateEnu>(inst->StateCurrent));

						for(unsigned short int i = 0; i < EM_MAX_AUDIT_ENTRIES; i++){
							strcpy(inst->Info.Last[EM_MAX_AUDIT_ENTRIES - i], inst->Info.Last[(EM_MAX_AUDIT_ENTRIES - 1) - i]);
						}
						sprintf(inst->Info.Last[0], "State: %s, time: %2.1f s.", oldStateStr, inst->Info.TimeInState);
					}

					inst->Info.TimeInState = 0;
					inst->Info.ParentName[0] = 0;
					inst->Info.ParentStateCurrent = STATE_UNDEFINED;
					inst->Info.ParentStateComplete = false;
					inst->Info.Level = 0;
					inst->Info.SiblingCount = 1;
					inst->StateCurrent = STATE_UNDEFINED;
					inst->SubState = 0;
					inst->StateInfo[0] = 0;
					memset(&inst->Command, 0, sizeof(inst->Command));
				}

			}
			break;
	}

}
```

#### ControlModule.cpp
```cpp
#include "BrdkPackML.h"
#include "../PackMLCore/PackMLModule.hpp"
#include "../PackMLCore/PackMLModuleTable.hpp"

extern unsigned long bur_heap_size;

extern PackMLModuleTable* pPackMLModuleTable;

// Main function. Is running cyclic together with FUB EquipmentModule()
void run(struct ControlModule* inst, PackMLModule* pPackMLModule)
{

	if (inst->Info.OnStateEntry){
		inst->Info.OnStateEntry = false;
	}
	if (inst->Info.OnSubStateEntry){
		inst->Info.OnSubStateEntry = false;
	}

	if(inst->Internal.oldSubState == -1){
		inst->SubState = -1;

		if(inst->Continue || !inst->Setup.StepMode){
			inst->Internal.oldSubState = inst->SubState = inst->Internal.nextSubState;
			inst->StateInfo[0] = 0;
			inst->Info.TimeInSubState = 0.0;
			inst->Info.OnSubStateEntry = true;
			inst->Internal.nextSubState = 0;
			inst->Continue = false;
		}
	} else if((inst->Internal.oldSubState != inst->SubState) && inst->State != -1){

		if(inst->Setup.AuditSubStateChange){

			for(unsigned short int i = 0; i < EM_MAX_AUDIT_ENTRIES; i++){
				strcpy(inst->Info.Last[EM_MAX_AUDIT_ENTRIES - i], inst->Info.Last[(EM_MAX_AUDIT_ENTRIES - 1) - i]);
			}
			sprintf(inst->Info.Last[0], "Substate: %ld, time: %2.1f s.", inst->Internal.oldSubState, inst->Info.TimeInSubState);
		}
		if(inst->Setup.StepMode && !inst->Continue){
			inst->Internal.nextSubState = inst->SubState;
			sprintf(inst->StateInfo, "Waiting for continue cmd. Next Substate: %ld", inst->Internal.nextSubState);
			inst->Info.TimeInSubState = 0.0;
			inst->Internal.oldSubState = inst->SubState = -1;
			inst->Continue = false;
		} else {
			inst->Internal.oldSubState = inst->SubState;
			inst->StateInfo[0] = 0;
			inst->Info.TimeInSubState = 0.0;
			inst->Info.OnSubStateEntry = true;
			inst->Continue = false;
		}
	}

	if(inst->Internal.oldState == -1){
		inst->State = -1;
		inst->SubState = 0;
		inst->Internal.oldSubState = 0;

		if(inst->Continue || !inst->Setup.StepMode){
			inst->Internal.oldState = inst->State = inst->Internal.nextState;
			inst->StateInfo[0] = 0;
			inst->Info.TimeInState = 0.0;
			inst->Info.TimeInSubState = 0.0;
			inst->Info.OnSubStateEntry = true;
			inst->Info.OnStateEntry = true;
			inst->Internal.nextState = 0;
			inst->Internal.nextSubState = 0;
			inst->Continue = false;
		}
	} else if (inst->State != inst->Internal.oldState){

		if(inst->Setup.AuditStateChange){

			for(unsigned short int i = 0; i < EM_MAX_AUDIT_ENTRIES; i++){
				strcpy(inst->Info.Last[EM_MAX_AUDIT_ENTRIES - i], inst->Info.Last[(EM_MAX_AUDIT_ENTRIES - 1) - i]);
			}
			sprintf(inst->Info.Last[0], "State: %ld, time: %2.1f s.", inst->Internal.oldState, inst->Info.TimeInState);
		}

		if(inst->Setup.StepMode && !inst->Continue){
			inst->Internal.nextState = inst->State;
			sprintf(inst->StateInfo, "Waiting for continue cmd. Next State: %ld", inst->Internal.nextState);
			inst->Info.TimeInState = 0.0;
			inst->Info.TimeInSubState = 0.0;
			inst->Internal.oldState = inst->State = -1;
			inst->Continue = false;
		} else {
			inst->Internal.oldState = inst->State;
			inst->SubState = 0;
			inst->Internal.oldSubState = 0;
			inst->StateInfo[0] = 0;
			inst->Info.TimeInState = 0.0;
			inst->Info.TimeInSubState = 0.0;
			inst->Info.OnStateEntry = true;
			inst->Info.OnSubStateEntry = true;
			inst->Continue = false;
		}
	}

	if (inst->Internal.oldParentState != inst->Info.ParentStateCurrent){
		inst->Continue = false;
		inst->Setup.StepMode = false;
	}

	inst->Internal.oldParentState = inst->Info.ParentStateCurrent;

	// Update the FB info
	// State info

	inst->Info.TimeInState += inst->Internal.cycleTime;
	inst->Info.TimeInSubState += inst->Internal.cycleTime;

	// Parent / Child / Sibling state/substate info
	if (pPackMLModule != nullptr){
		inst->Info.Level = pPackMLModule->getHierarchyLevel() + 1;
		inst->Info.ParentStateCurrent = static_cast<EMPackMLStateEnum>(pPackMLModule->getCurrentState());
	} else {
		inst->Info.Level = 0;
		inst->Info.ParentStateCurrent = STATE_UNDEFINED;
	}

	if(inst->Interface.Enable){
		inst->Internal.oldPubSubEnable = true;

		for(unsigned short int i = 0; i < EM_MAX_SUBSCRIPTIONS + 1; i++){

			if(inst->Interface.SubscriptionValid[i]){
				memcpy(reinterpret_cast<EMUserDataPubSubType*>(&inst->Interface.Subscribe[i]), reinterpret_cast<EMUserDataPubSubType*>(inst->Internal.subscriptionUserDataAddress[i]), sizeof(EMUserDataPubSubType));
			}

			if(strcmp(inst->Interface.SubscriptionEMName[i], inst->Internal.subscribedToEMName[i]) != 0){
				PackMLModule* pSubscribtionEm = pPackMLModuleTable->getModuleByName(inst->Interface.SubscriptionEMName[i]);
				if(pSubscribtionEm != nullptr){
					inst->Internal.subscriptionUserDataAddress[i] = reinterpret_cast<unsigned long int>(pSubscribtionEm->getUserMemoryPtr());
					inst->Interface.SubscriptionValid[i] = true;
					strcpy(inst->Internal.subscribedToEMName[i], inst->Interface.SubscriptionEMName[i]);
				} else {
					inst->Interface.SubscriptionValid[i] = false;
					inst->Internal.subscriptionUserDataAddress[i] = 0;
					inst->Internal.subscribedToEMName[i][0] = 0;
				}

				memset(reinterpret_cast<EMUserDataPubSubType*>(&inst->Interface.Subscribe[i]), 0, sizeof(EMUserDataPubSubType));

			}

		}
	} else if(not inst->Interface.Enable && inst->Internal.oldPubSubEnable){
		inst->Internal.oldPubSubEnable = false;
		memset(reinterpret_cast<EMUserDataPubSubType*>(&inst->Interface.Subscribe), 0, sizeof(EMUserDataPubSubType) * (EM_MAX_SUBSCRIPTIONS + 1));
		memset(reinterpret_cast<bool*>(&inst->Interface.SubscriptionValid), 0, sizeof(bool) * (EM_MAX_SUBSCRIPTIONS + 1));
		memset(reinterpret_cast<unsigned long int*>(&inst->Internal.subscriptionUserDataAddress), 0, sizeof(unsigned long int) * (EM_MAX_SUBSCRIPTIONS + 1));
		memset(reinterpret_cast<char*>(&inst->Internal.subscribedToEMName), 0, 256 * (EM_MAX_SUBSCRIPTIONS + 1));
	}

}

// ------------ IEC Functions and Function Blocks -----------------------------------------

void ControlModule(struct ControlModule* inst)
{

	// Initialize the module
	switch(inst->Internal.state){

		case 0:
			{
				// get name
				if(strlen(inst->Setup.Name) == 0){
					ST_name(0, inst->Setup.Name, 0);
				}

				char moduleName[256] = {""};

				if (inst->Setup.NameIndex == EM_MAX_NAME_INDEX){
					strcpy(moduleName, inst->Setup.Name);
				} else {
					sprintf(moduleName, "%s%d", inst->Setup.Name, inst->Setup.NameIndex);
				}

				strcpy(inst->Info.CmName, moduleName);

				RTInfo_typ RTInfo_0;
				RTInfo_0.enable = 1;
				RTInfo(&RTInfo_0);
				inst->Internal.cycleTime = static_cast<float>(RTInfo_0.cycle_time) * 0.000001;
				inst->Info.CycleTime = inst->Internal.cycleTime;
				inst->Internal.state = 30;
			}
			break;

		case 30: // Init EM phase // interlinking
			{
				if(strlen(inst->Setup.ParentName) > 0){
					inst->Internal.state = 35;
				} else {
					inst->Internal.state = 40;
				}
				strcpy(inst->Info.ParentName, inst->Setup.ParentName);
			}
			break;

		case 35:
			{

				PackMLModule* pPackMLModule = pPackMLModuleTable->getModuleByName(inst->Info.ParentName);

				if(strcmp(inst->Setup.ParentName, inst->Info.ParentName) != 0){
					inst->Internal.state = 30;

				} else if(pPackMLModule != nullptr){
					inst->Internal.parentEmAddress = reinterpret_cast<unsigned long int>(pPackMLModule);
					inst->Info.ParentEmAddress = inst->Internal.parentEmAddress;
					inst->Info.ParentEmIndex = pPackMLModuleTable->getModuleIndexByName(inst->Info.ParentName);
					inst->Internal.state = 40;
				}

			}
			break;

		case 40: // run state
			// if EmLinkParent changes reinitilise the module in state 30
			{
				PackMLModule* pPackMLModule = reinterpret_cast<PackMLModule*>(inst->Internal.parentEmAddress);

				if(strcmp(inst->Setup.ParentName, inst->Info.ParentName) != 0){
					inst->Info.ParentName[0] = 0;
					inst->Info.ParentEmAddress = 0;
					inst->Info.ParentEmIndex = 0;
					inst->Internal.parentEmAddress = 0;
					inst->Internal.state = 30;
				}
				run(inst, pPackMLModule);
			}
			break;
	}

}
```

### Library Logical/Libraries/PackMLCore (ANSIC, version 2.0.3)

#### PackMLModule.hpp
```cpp
#ifndef __PACKMLMODULE_HPP__
#define __PACKMLMODULE_HPP__

#include "PackMLModuleEnums.hpp"
#include <vector>
#include <string>
#include <string.h>
//#include <cmath>
#include "AtomicSemaphore.hpp"
#include "PackMLModuleSharedInfo.hpp"

		// PackMLModule main class
class PackMLModule {

	public:
	PackMLModule(const char* pModuleName);
	~PackMLModule();

	// *** onCreated() ***
	// root module
	void initModule();
	// child module
	bool initModule(PackMLModule* pParent);

	// *** onBeforeShutdown() ***
	bool exitModule();

	// *** run() ***
	void runPackMLModule();

	// **********************************************************
	// ************* Real time parameter update *****************
	// **********************************************************
	void setActivationCondition(short int newParameter){
		activationCondition_ = newParameter;
	}

	void setOverrideAbort(bool newParameter)
	{
		overrideAbort_ = newParameter && (hierarchyLevel_ > 0);
	}
	void setOverrideStop(bool newParameter)
	{
		overrideStop_ = newParameter && (hierarchyLevel_ > 0);
	}
	void setOverrideClear(bool newParameter)
	{
		overrideClear_ = newParameter && (hierarchyLevel_ > 0);
	}
	void setOverrideReset(bool newParameter)
	{
		overrideReset_ = newParameter && (hierarchyLevel_ > 0);
	}
	void setOverrideStart(bool newParameter)
	{
		overrideStart_ = newParameter && (hierarchyLevel_ > 0);
	}
	void setOverrideSuspend(bool newParameter)
	{
		overrideSuspend_ = newParameter && (hierarchyLevel_ > 0);
	}
	void setOverrideUnsuspend(bool newParameter)
	{
		overrideUnsuspend_ = newParameter && (hierarchyLevel_ > 0);
	}
	void setOverrideHold(bool newParameter)
	{
		overrideHold_ = newParameter && (hierarchyLevel_ > 0);
	}
	void setOverrideUnhold(bool newParameter)
	{
		overrideUnhold_ = newParameter && (hierarchyLevel_ > 0);
	}
	void setOverrideComplete(bool newParameter)
	{
		overrideComplete_ = newParameter && (hierarchyLevel_ > 0);
	}

	void setReactToAbort(bool newParameter)
	{
		reactToAbort_ = newParameter && (hierarchyLevel_ > 0);
	}
	void setReactToStop(bool newParameter)
	{
		reactToStop_ = newParameter && (hierarchyLevel_ > 0);
	}
	void setReactToClear(bool newParameter)
	{
		reactToClear_ = newParameter && (hierarchyLevel_ > 0);
	}
	void setReactToReset(bool newParameter)
	{
		reactToReset_ = newParameter && (hierarchyLevel_ > 0);
	}
	void setReactToStart(bool newParameter)
	{
		reactToStart_ = newParameter && (hierarchyLevel_ > 0);
	}
	void setReactToSuspend(bool newParameter)
	{
		reactToSuspend_ = newParameter && (hierarchyLevel_ > 0);
	}
	void setReactToUnsuspend(bool newParameter)
	{
		reactToUnsuspend_ = newParameter && (hierarchyLevel_ > 0);
	}
	void setReactToHold(bool newParameter)
	{
		reactToHold_ = newParameter && (hierarchyLevel_ > 0);
	}
	void setReactToUnhold(bool newParameter)
	{
		reactToUnhold_ = newParameter && (hierarchyLevel_ > 0);
	}
	void setReactToComplete(bool newParameter)
	{
		reactToComplete_ = newParameter && (hierarchyLevel_ > 0);
	}

	void setEscalateAbort(bool newParameter)
	{
		escalateAbort_ = newParameter && (hierarchyLevel_ > 0);
	}
	void setEscalateStop(bool newParameter)
	{
		escalateStop_ = newParameter && (hierarchyLevel_ > 0);
	}
	void setEscalateClear(bool newParameter)
	{
		escalateClear_ = newParameter && (hierarchyLevel_ > 0);
	}
	void setEscalateReset(bool newParameter)
	{
		escalateReset_ = newParameter && (hierarchyLevel_ > 0);
	}
	void setEscalateStart(bool newParameter)
	{
		escalateStart_ = newParameter && (hierarchyLevel_ > 0);
	}
	void setEscalateSuspend(bool newParameter)
	{
		escalateSuspend_ = newParameter && (hierarchyLevel_ > 0);
	}
	void setEscalateUnsuspend(bool newParameter)
	{
		escalateUnsuspend_ = newParameter && (hierarchyLevel_ > 0);
	}
	void setEscalateHold(bool newParameter)
	{
		escalateHold_ = newParameter && (hierarchyLevel_ > 0);
	}
	void setEscalateUnhold(bool newParameter)
	{
		escalateUnhold_ = newParameter && (hierarchyLevel_ > 0);
	}
	void setEscalateComplete(bool newParameter)
	{
		escalateComplete_ = newParameter && (hierarchyLevel_ > 0);
	}

	bool evaluateCmdAbort(bool& newCmd);
	bool evaluateCmdStop(bool& newCmd);
	bool evaluateCmdClear(bool& newCmd);
	bool evaluateCmdReset(bool& newCmd);
	bool evaluateCmdStart(bool& newCmd);
	bool evaluateCmdSuspend(bool& newCmd);
	bool evaluateCmdUnsuspend(bool& newCmd);
	bool evaluateCmdHold(bool& newCmd);
	bool evaluateCmdUnhold(bool& newCmd);
	bool evaluateCmdComplete(bool& newCmd);
	bool evaluateCmdStateComplete(bool& newCmd);

	bool setCmdAbort();
	bool setCmdStop();
	bool setCmdClear();
	bool setCmdReset();
	bool setCmdStart();
	bool setCmdSuspend();
	bool setCmdUnsuspend();
	bool setCmdHold();
	bool setCmdUnhold();
	bool setCmdComplete();
	bool setCmdStateComplete();

	bool getCmdAbort(){
		return abort_;
	}
	bool getCmdStop(){
		return stop_;
	}
	bool getCmdClear(){
		return clear_;
	}
	bool getCmdReset(){
		return reset_;
	}
	bool getCmdStart(){
		return start_;
	}
	bool getCmdSuspend(){
		return suspend_;
	}
	bool getCmdUnsuspend(){
		return unsuspend_;
	}
	bool getCmdHold(){
		return hold_;
	}
	bool getCmdUnhold(){
		return unhold_;
	}
	bool getCmdComplete(){
		return complete_;
	}
	bool getCmdStateComplete(){
		return stateComplete_;
	}

	void resetCmdAbort();
	void resetCmdStop();
	void resetCmdClear();
	void resetCmdReset();
	void resetCmdStart();
	void resetCmdSuspend();
	void resetCmdUnsuspend();
	void resetCmdHold();
	void resetCmdUnhold();
	void resetCmdComplete();
	void resetCmdStateComplete();

	// **********************************************************

	PackMLModuleStateEnu getParentCurrentState();

	long int getParentCurrentSubState();

	const char *getParentName();

	bool getParentStateComplete();

	PackMLModule* getParentAdr() { return pParentLink_; }

	bool getSiblingsStateComplete();

	bool getChildrenStateComplete();

	const char *getCurrentStateStr() const;

	const char *getStateStr(PackMLModuleStateEnu state) const;

	const char *getCurrentModeStr() const;

	unsigned long getChildCount() { return childCount_; }

	unsigned long getSiblingCount();

	unsigned short getHierarchyLevel()
	{
		return hierarchyLevel_;
	}

	// ************************* Service interface methods *********************
	// Name of the module
	const char* getModuleName() { return moduleName_.c_str(); }
	unsigned long int getModuleId() { return moduleId_; }

	// Called by the IEC function
	const char* getStateInfo() { return stateInfo_.c_str(); }

	bool setCurrentMode(long int mode);
	long int getCurrentMode(){ return modeCurrent_; }
	const char* getCurrentModeName() const;
	const char* getModeName(signed long int modeId) const;
	bool isModeChangePossible();

	bool getModuleReady() { return moduleReady_; }
	void setModuleReady(bool value);

	void setNewModeCurrent(long int mode);
	void setHierarchyLevel(unsigned short level);
	void setAllStateComplete();

	bool registerChild(PackMLModule* pChild); // called during onCreated()
	bool unregisterChild(PackMLModule* pChild);

	void escalateCmdAbort();
	void escalateCmdClear();

	void escalateCmdSuspend();
	void escalateCmdUnsuspend();

	void escalateCmdHold();
	void escalateCmdUnhold();

	void escalateCmdStop();
	void escalateCmdReset();

	void escalateCmdStart();
	void escalateCmdComplete();

	void propagateCmdAbort(bool root);
	void propagateCmdClear(bool root);

	void propagateCmdSuspend(bool root);
	void propagateCmdUnsuspend(bool root);

	void propagateCmdHold(bool root);
	void propagateCmdUnhold(bool root);

	void propagateCmdStop(bool root);
	void propagateCmdReset(bool root);

	void propagateCmdStart(bool root);
	void propagateCmdComplete(bool root);

	PackMLModuleStateEnu getCurrentState(){
		return stateCurrent_;
	}

	void setCurrentSubState(long int subState){
		subStateCurrent_ = subState;
		timeInSubState_ = 0.0;
	}

	long int getCurrentSubState(){
		return subStateCurrent_;
	}

	bool getStateComplete(){
		return stateComplete_;
	}
	// check if child wants to be synchronized
	bool needParentSynch(PackMLModuleStateEnu parentState);

	void setActivationPv(bool activationPv) { activationPv_ = activationPv; }

	unsigned long int getWaitingForIndex() {
		return waitingForIndex_;
	}

	unsigned long int getInterruptedByIndex() {
		return interruptedByIndex_;
	}

	PackMLModuleStateEnu getInterruptedInState() {
		return interruptedInState_;
	}

	signed long int getInterruptedInSubState() {
		return interruptedInSubState_;
	}

	PackMLModuleStateEnu getChildCurrentState(unsigned long int childIndex);
	long int getChildCurrentSubState(unsigned long int childIndex);
	bool getChildStateComplete(unsigned long int childIndex);
	const char* getChildName(unsigned long int childIndex);

	PackMLModuleStateEnu getSiblingCurrentState(unsigned long int siblingIndex);
	long int getSiblingCurrentSubState(unsigned long int siblingIndex);
	bool getSiblingStateComplete(unsigned long int siblingIndex);
	const char* getSiblingName(unsigned long int siblingIndex);

	float getTimeInState() { return timeInState_; }
	float getTimeInSubState() { return timeInSubState_; }

	void setCycleTime(float cycleTime) { cycleTime_ = cycleTime; }

	PackMLModule* getParentPtr();
	PackMLModule* getChildPtr(unsigned long int childIdx);
	PackMLModule* getSiblingPtr(unsigned long int siblingIdx);

	void* createUserMemory(unsigned long int userMemorySize);
	void* getUserMemoryPtr();
	void deleteUserMemory();

	bool isActingState(PackMLModuleStateEnu state);
	bool isWaitingState(PackMLModuleStateEnu state){
		return !isActingState(state);
	}

	void setInterruptedBy(PackMLModule* pPackMLModule, PackMLModuleStateEnu cmdState);

	void setStateInfo(std::string stateInfo){
		stateInfo_ = stateInfo;
	}

	void setModuleIndex(unsigned long int index){
		moduleIndex_ = index;
	}

	unsigned long int getModuleIndex(){
		return moduleIndex_;
	}

	void escalateInterruptedBy(unsigned long int moduleIndex, PackMLModuleStateEnu state, signed long int subState, PackMLModuleStateEnu cmdState);
	void propagateInterruptedBy(unsigned long int moduleIndex, PackMLModuleStateEnu state, signed long int subState, PackMLModuleStateEnu cmdState, bool root);
	void escalateWaitingFor(unsigned long int waitingForIndex, unsigned short int waitingForLevel, PackMLModuleStateEnu cmdState);
	void escalateResetWaitingFor(unsigned long int waitingForIndex);

	private:

	// --------------------------------------------------------
	// **************** Will be private ***********************
	// --------------------------------------------------------

	// unique service name identifier
	std::string moduleName_;
	unsigned long moduleId_;
	unsigned long int moduleIndex_;
	unsigned long generateId_(const char *pName);

	// used during the registration
	AtomicSemaphore semaphore_;

	// **************** FB parameters placeholder ******************
	std::string stateInfo_;

	short int activationCondition_;

	bool overrideAbort_;
	bool overrideStop_;
	bool overrideClear_;
	bool overrideReset_;
	bool overrideStart_;
	bool overrideSuspend_;
	bool overrideUnsuspend_;
	bool overrideHold_;
	bool overrideUnhold_;
	bool overrideComplete_;

	bool reactToAbort_;
	bool reactToStop_;
	bool reactToClear_;
	bool reactToReset_;
	bool reactToStart_;
	bool reactToSuspend_;
	bool reactToUnsuspend_;
	bool reactToHold_;
	bool reactToUnhold_;
	bool reactToComplete_;

	bool escalateAbort_;
	bool escalateStop_;
	bool escalateClear_;
	bool escalateReset_;
	bool escalateStart_;
	bool escalateSuspend_;
	bool escalateUnsuspend_;
	bool escalateHold_;
	bool escalateUnhold_;
	bool escalateComplete_;

	// ****************** Hierarchy related stuff ***********************

	// Pointers to the parent/childs in the hierarchy
	// Change it to smart pointers
	PackMLModule* pParentLink_;
	std::vector<PackMLModule*> childLinks_;
	unsigned long int parentLinkAdr_;

	// Configure the hierarchy
	bool linkToParent_(PackMLModule* pParent);
	bool unlinkFromParent_();

	bool hasParent_;
	unsigned long childCount_;
	unsigned short hierarchyLevel_;

	bool moduleReady_;

	// *************** PackML State Manager *******************
	long int modeCurrent_;
	PackMLModuleStateEnu stateCurrent_;
	long int subStateCurrent_;

	bool activate_;
	bool deactivate_;

	// Internal cmds
	bool abort_;
	bool clear_;
	bool stop_;
	bool reset_;
	bool start_;
	bool hold_;
	bool unhold_;
	bool suspend_;
	bool unsuspend_;
	bool complete_;
	bool stateComplete_;

	bool oldAbort_;
	bool oldClear_;
	bool oldStop_;
	bool oldReset_;
	bool oldStart_;
	bool oldHold_;
	bool oldUnhold_;
	bool oldSuspend_;
	bool oldUnsuspend_;
	bool oldComplete_;
	bool oldStateComplete_;

	bool externalAbort_;
	bool externalClear_;
	bool externalStop_;
	bool externalReset_;
	bool externalStart_;
	bool externalHold_;
	bool externalUnhold_;
	bool externalSuspend_;
	bool externalUnsuspend_;
	bool externalComplete_;
	bool externalStateComplete_;

	void updatePackMLModel_();

	void checkActivationCondition_();

	void checkParentStateCondition_();

	bool setCmd_(PackMLModuleStateEnu targetActingState);
	void resetCmd_(PackMLModuleStateEnu targetActingState);

	void executeCmd_(PackMLModuleStateEnu targetState);

	void executeActingState_(PackMLModuleStateEnu targetState);

	bool stateExistInPattern_(unsigned long stateBitPattern,
	PackMLModuleStateEnu state);

	bool cmdValid_(PackMLModuleStateEnu state);
	// Checks if the all the children are in the provided state
	bool childrenInState_(PackMLModuleStateEnu state);
	// Checks if the children are in need of synchronization for the provided
	// state
	bool childrenInSynch_(PackMLModuleStateEnu targetState);

	bool isChild_(PackMLModule* pModule);

	// Reset the cmds, substate, status etc when a state changes
	void resetInternalCmds_();

	// Waiting for and aborted by related stuff
	void setWaitingFor_(PackMLModuleStateEnu cmdState);
	void resetWaitingFor_();

	void setInterruptedBy_(PackMLModuleStateEnu cmdState);
	void resetInterruptedBy_();

	unsigned long int waitingForIndex_;
	unsigned short waitingForLevel_;

	unsigned long int interruptedByIndex_;
	PackMLModuleStateEnu interruptedInState_;
	signed long int interruptedInSubState_;

	bool activationPv_;
	float timeInState_;
	float timeInSubState_;
	float cycleTime_; // ms

	void updateTimeInState_() {
		timeInState_ += cycleTime_;
		timeInSubState_ += cycleTime_;
	}

	void* pUserData_;
	unsigned long int userDataSize_;

};

#endif // __MAPP_MXPACKML_PACKMLMODULE_HPP__
```

#### PackMLModule.cpp
```cpp
#include "PackMLModule.hpp"

		// -----------------------------------------------------------------------------

PackMLModule::PackMLModule(const char* pModuleName) : moduleName_(pModuleName),
	moduleId_(0),
	moduleIndex_(0xFFFFFFFF),
	semaphore_(),
	activationCondition_(0),
	overrideAbort_(false),
	overrideStop_(false),
	overrideClear_(false),
	overrideReset_(false),
	overrideStart_(false),
	overrideSuspend_(false),
	overrideUnsuspend_(false),
	overrideHold_(false),
	overrideUnhold_(false),
	overrideComplete_(false),
	reactToAbort_(false),
	reactToStop_(false),
	reactToClear_(false),
	reactToReset_(false),
	reactToStart_(false),
	reactToSuspend_(false),
	reactToUnsuspend_(false),
	reactToHold_(false),
	reactToUnhold_(false),
	reactToComplete_(false),
	escalateAbort_(false),
	escalateStop_(false),
	escalateClear_(false),
	escalateReset_(false),
	escalateStart_(false),
	escalateSuspend_(false),
	escalateUnsuspend_(false),
	escalateHold_(false),
	escalateUnhold_(false),
	escalateComplete_(false),
	pParentLink_(nullptr),
	childLinks_(),
	parentLinkAdr_(0),
	hasParent_(false),
	childCount_(0),
	hierarchyLevel_(0),
	moduleReady_(false),
	modeCurrent_(1),
	stateCurrent_(ST_UNDEFINED),
	subStateCurrent_(0),
	activate_(false),
	deactivate_(false),
	abort_(false),
	clear_(false),
	stop_(false),
	reset_(false),
	start_(false),
	hold_(false),
	unhold_(false),
	suspend_(false),
	unsuspend_(false),
	complete_(false),
	stateComplete_(false),
	oldAbort_(false),
	oldClear_(false),
	oldStop_(false),
	oldReset_(false),
	oldStart_(false),
	oldHold_(false),
	oldUnhold_(false),
	oldSuspend_(false),
	oldUnsuspend_(false),
	oldComplete_(false),
	oldStateComplete_(false),
	externalAbort_(false),
	externalClear_(false),
	externalStop_(false),
	externalReset_(false),
	externalStart_(false),
	externalHold_(false),
	externalUnhold_(false),
	externalSuspend_(false),
	externalUnsuspend_(false),
	externalComplete_(false),
	externalStateComplete_(false),
	waitingForIndex_(0xFFFFFFFF),
	waitingForLevel_(0),
	interruptedByIndex_(0xFFFFFFFF),
	interruptedInState_(ST_UNDEFINED),
	activationPv_(false),
	timeInState_(0.0),
	timeInSubState_(0.0),
	cycleTime_(0.0),
	pUserData_(nullptr),
	userDataSize_(0)
{
	//	moduleName_ = "";
	stateInfo_ = "";
	moduleId_ = generateId_(pModuleName);

}

		// -----------------------------------------------------------------------------

PackMLModule::~PackMLModule()
{
	free(pUserData_);
}

// -----------------------------------------------------------------------------
void* PackMLModule::createUserMemory(unsigned long int userMemorySize){
	if(pUserData_ != nullptr)
		return pUserData_;

	pUserData_ = calloc(userMemorySize, sizeof(char));
	userDataSize_ = userMemorySize;
//	memset(pUserData_, 0, userDataSize_);

	return pUserData_;
}
// -----------------------------------------------------------------------------
void* PackMLModule::getUserMemoryPtr(){
	return pUserData_;
}

void PackMLModule::deleteUserMemory(){
	free(pUserData_);
}

// -----------------------------------------------------------------------------

void PackMLModule::initModule()
{
	setNewModeCurrent(modeCurrent_);
	setHierarchyLevel(0);
	setModuleReady(true);

}

bool PackMLModule::initModule(PackMLModule* pParent)
{
	if(pParent == nullptr || pParent == this || isChild_(pParent)){
		return false;
	}
	return linkToParent_(pParent);
}

		// -----------------------------------------------------------------------------
bool PackMLModule::exitModule()
{
	// decide what to do here, do we need to reset those when unlinking from parent
	resetWaitingFor_();
	resetInterruptedBy_();

	// ******
	// nested call for resetWaitingFor and InterruptedBy for all children and childrens children
	// ******

	setNewModeCurrent(modeCurrent_);
	setHierarchyLevel(0);
	setModuleReady(false);

	stateInfo_ = "";

	overrideAbort_ = false;
	overrideStop_ = false;
	overrideClear_ = false;
	overrideReset_ = false;
	overrideStart_ = false;
	overrideSuspend_ = false;
	overrideUnsuspend_ = false;
	overrideHold_ = false;
	overrideUnhold_ = false;
	overrideComplete_ = false;
	reactToAbort_ = false;
	reactToStop_ = false;
	reactToClear_ = false;
	reactToReset_ = false;
	reactToStart_ = false;
	reactToSuspend_ = false;
	reactToUnsuspend_ = false;
	reactToHold_ = false;
	reactToUnhold_ = false;
	reactToComplete_ = false;
	escalateAbort_ = false;
	escalateStop_ = false;
	escalateClear_ = false;
	escalateReset_ = false;
	escalateStart_ = false;
	escalateSuspend_ = false;
	escalateUnsuspend_ = false;
	escalateHold_ = false;
	escalateUnhold_ = false;
	escalateComplete_ = false;
	activate_ = false;
	deactivate_ = false;

	resetInternalCmds_();

	if(!hasParent_){
		return true;
	}
	return unlinkFromParent_();
}

		// -----------------------------------------------------------------------------

void PackMLModule::runPackMLModule()
{
	updateTimeInState_();
	// check parent state condition
	checkParentStateCondition_();
	// update the packml model
	updatePackMLModel_();

}
		// ---------------------------------------------------------------------------

		// called during onCreated() if parent found and in onService()
bool PackMLModule::linkToParent_(PackMLModule* pParent)
{
	if(pParent->registerChild(this)){
		pParentLink_ = pParent;
		hasParent_ = true;
		return true;
	}
	return false;
}

		// -------------------------------------------------------------------------

bool PackMLModule::unlinkFromParent_()
{
	if(pParentLink_->unregisterChild(this)){
		pParentLink_ = nullptr;
		hasParent_ = false;
		return true;
	}
	return false;
}

		// -------------------------------------------------------------------------

bool PackMLModule::registerChild(PackMLModule* pChild)
{

	if(isChild_(pChild))
		return true;

	if(!semaphore_.acquire())
		return false;

	childLinks_.push_back(pChild);

	pChild->setNewModeCurrent(modeCurrent_);
	pChild->setHierarchyLevel(hierarchyLevel_ + 1);
	pChild->setModuleReady(moduleReady_);

	childCount_ = childLinks_.size();
	semaphore_.release();
	return true;
}

		// -------------------------------------------------------------------------

bool PackMLModule::unregisterChild(PackMLModule* pChild)
{
	//			BR::Core::MutexLocker lock(&mutex_);

	if(!semaphore_.acquire())
		return false;

	for (unsigned short i = 0; i < childCount_; ++i) {
		if (childLinks_[i]->getModuleId() == pChild->getModuleId()) {
			childLinks_.erase(childLinks_.begin() + i);
			break;
		}
	}

	childCount_ = childLinks_.size();
	semaphore_.release();
	return true;
}

		// -------------------------------------------------------------------------

void PackMLModule::setModuleReady(bool value)
{
	moduleReady_ = value;

	if (moduleReady_) {
		stateCurrent_ = ST_DEACTIVATED;
	}
	else {
		stateCurrent_ = ST_UNDEFINED;
	}

	for (unsigned short i = 0; i < childCount_; ++i) {
		childLinks_[i]->setModuleReady(value);
	}
}

void PackMLModule::setHierarchyLevel(unsigned short level)
{
	hierarchyLevel_ = level;

	for (unsigned short i = 0; i < childCount_; ++i) {
		childLinks_[i]->setHierarchyLevel(level + 1);
	}

}

void PackMLModule::setAllStateComplete()
{
	stateComplete_ = true;
	externalStateComplete_ = stateComplete_;

	for (unsigned short i = 0; i < childCount_; ++i) {
		childLinks_[i]->setAllStateComplete();
	}

}

		// -------------------------------------------------------------------------

unsigned long PackMLModule::generateId_(const char *pName)
{
	unsigned long int N = strlen(pName);
	unsigned long int b    = 378551;
	unsigned long int a    = 63689;
	unsigned long int hash = 0;

	for(std::size_t i = 0; i < N; i++)
	{
		hash = hash * a + pName[i];
		a    = a * b;
	}

	return (hash & 0x7FFFFFFF);
}
```
